// TIA Portal V20 export
FUNCTION_BLOCK "Simulation"   // FB112, LAD
// stored: MemoryReserve 100, Namespace Unit1.Em5, SetENOAutomatically false
   VAR_INPUT
      simulation : Bool;
   END_VAR
   VAR
      Simulation_addon_Instance { S7_SetPoint := 'True'} : "Simulation_addon";
      Simulation_addon_Instance_1 { S7_SetPoint := 'True'} : "Simulation_addon";
      Simulation_addon_Instance_2 { S7_SetPoint := 'True'} : "Simulation_addon";
      Simulation_addon_Instance_3 { S7_SetPoint := 'True'} : "Simulation_addon";
   END_VAR
BEGIN

REGION Network 1: cmNgAndManualInputCylinderUpDown
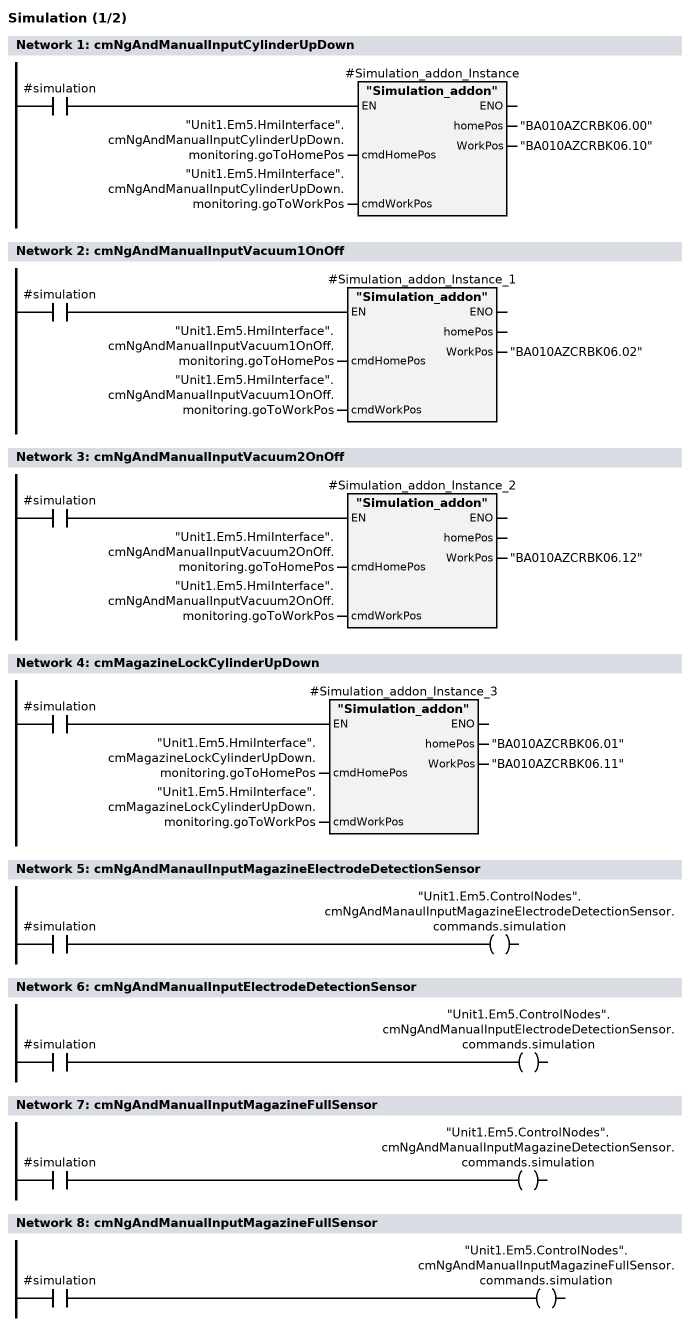
   RUNG wire#powerrail
      Contact( #simulation )
      #Simulation_addon_Instance(cmdHomePos := "Unit1.Em5.HmiInterface".cmNgAndManualInputCylinderUpDown.monitoring.goToHomePos, cmdWorkPos := "Unit1.Em5.HmiInterface".cmNgAndManualInputCylinderUpDown.monitoring.goToWorkPos, homePos => "BA010AZCRBK06.00", WorkPos => "BA010AZCRBK06.10")
   END_RUNG
   // the same network as SCL:
   IF #simulation THEN
       #Simulation_addon_Instance(cmdHomePos := "Unit1.Em5.HmiInterface".cmNgAndManualInputCylinderUpDown.monitoring.goToHomePos,   // "Simulation_addon"
                               cmdWorkPos := "Unit1.Em5.HmiInterface".cmNgAndManualInputCylinderUpDown.monitoring.goToWorkPos,
                               homePos => "BA010AZCRBK06.00",
                               WorkPos => "BA010AZCRBK06.10");
   END_IF;
END_REGION

REGION Network 2: cmNgAndManualInputVacuum1OnOff
   RUNG wire#powerrail
      Contact( #simulation )
      #Simulation_addon_Instance_1(cmdHomePos := "Unit1.Em5.HmiInterface".cmNgAndManualInputVacuum1OnOff.monitoring.goToHomePos, cmdWorkPos := "Unit1.Em5.HmiInterface".cmNgAndManualInputVacuum1OnOff.monitoring.goToWorkPos, homePos =>, WorkPos => "BA010AZCRBK06.02")
   END_RUNG
   // the same network as SCL:
   IF #simulation THEN
       #Simulation_addon_Instance_1(cmdHomePos := "Unit1.Em5.HmiInterface".cmNgAndManualInputVacuum1OnOff.monitoring.goToHomePos,   // "Simulation_addon"
                               cmdWorkPos := "Unit1.Em5.HmiInterface".cmNgAndManualInputVacuum1OnOff.monitoring.goToWorkPos,
                               WorkPos => "BA010AZCRBK06.02");
   END_IF;
END_REGION

REGION Network 3: cmNgAndManualInputVacuum2OnOff
   RUNG wire#powerrail
      Contact( #simulation )
      #Simulation_addon_Instance_2(cmdHomePos := "Unit1.Em5.HmiInterface".cmNgAndManualInputVacuum2OnOff.monitoring.goToHomePos, cmdWorkPos := "Unit1.Em5.HmiInterface".cmNgAndManualInputVacuum2OnOff.monitoring.goToWorkPos, homePos =>, WorkPos => "BA010AZCRBK06.12")
   END_RUNG
   // the same network as SCL:
   IF #simulation THEN
       #Simulation_addon_Instance_2(cmdHomePos := "Unit1.Em5.HmiInterface".cmNgAndManualInputVacuum2OnOff.monitoring.goToHomePos,   // "Simulation_addon"
                               cmdWorkPos := "Unit1.Em5.HmiInterface".cmNgAndManualInputVacuum2OnOff.monitoring.goToWorkPos,
                               WorkPos => "BA010AZCRBK06.12");
   END_IF;
END_REGION

REGION Network 4: cmMagazineLockCylinderUpDown
   RUNG wire#powerrail
      Contact( #simulation )
      #Simulation_addon_Instance_3(cmdHomePos := "Unit1.Em5.HmiInterface".cmMagazineLockCylinderUpDown.monitoring.goToHomePos, cmdWorkPos := "Unit1.Em5.HmiInterface".cmMagazineLockCylinderUpDown.monitoring.goToWorkPos, homePos => "BA010AZCRBK06.01", WorkPos => "BA010AZCRBK06.11")
   END_RUNG
   // the same network as SCL:
   IF #simulation THEN
       #Simulation_addon_Instance_3(cmdHomePos := "Unit1.Em5.HmiInterface".cmMagazineLockCylinderUpDown.monitoring.goToHomePos,   // "Simulation_addon"
                               cmdWorkPos := "Unit1.Em5.HmiInterface".cmMagazineLockCylinderUpDown.monitoring.goToWorkPos,
                               homePos => "BA010AZCRBK06.01",
                               WorkPos => "BA010AZCRBK06.11");
   END_IF;
END_REGION

REGION Network 5: cmNgAndManaulInputMagazineElectrodeDetectionSensor
   RUNG wire#powerrail
      Contact( #simulation )
      Coil( "Unit1.Em5.ControlNodes".cmNgAndManaulInputMagazineElectrodeDetectionSensor.commands.simulation )
   END_RUNG
   // the same network as SCL:
   "Unit1.Em5.ControlNodes".cmNgAndManaulInputMagazineElectrodeDetectionSensor.commands.simulation := #simulation;
END_REGION

REGION Network 6: cmNgAndManualInputElectrodeDetectionSensor
   RUNG wire#powerrail
      Contact( #simulation )
      Coil( "Unit1.Em5.ControlNodes".cmNgAndManualInputElectrodeDetectionSensor.commands.simulation )
   END_RUNG
   // the same network as SCL:
   "Unit1.Em5.ControlNodes".cmNgAndManualInputElectrodeDetectionSensor.commands.simulation := #simulation;
END_REGION

REGION Network 7: cmNgAndManualInputMagazineFullSensor
   RUNG wire#powerrail
      Contact( #simulation )
      Coil( "Unit1.Em5.ControlNodes".cmNgAndManualInputMagazineDetectionSensor.commands.simulation )
   END_RUNG
   // the same network as SCL:
   "Unit1.Em5.ControlNodes".cmNgAndManualInputMagazineDetectionSensor.commands.simulation := #simulation;
END_REGION

REGION Network 8: cmNgAndManualInputMagazineFullSensor
   RUNG wire#powerrail
      Contact( #simulation )
      Coil( "Unit1.Em5.ControlNodes".cmNgAndManualInputMagazineFullSensor.commands.simulation )
   END_RUNG
   // the same network as SCL:
   "Unit1.Em5.ControlNodes".cmNgAndManualInputMagazineFullSensor.commands.simulation := #simulation;
END_REGION

REGION Network 9: cmMagazineSafetyPinIdlePosition
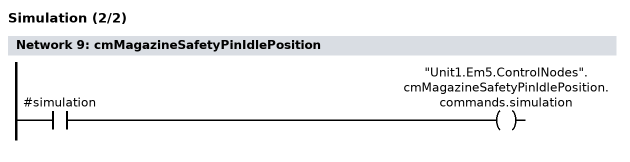
   RUNG wire#powerrail
      Contact( #simulation )
      Coil( "Unit1.Em5.ControlNodes".cmMagazineSafetyPinIdlePosition.commands.simulation )
   END_RUNG
   // the same network as SCL:
   "Unit1.Em5.ControlNodes".cmMagazineSafetyPinIdlePosition.commands.simulation := #simulation;
END_REGION
END_FUNCTION_BLOCK
